// TIA Portal V18 export
// export: Created 2025-12-01T17:50:36.3947Z, ExportSetting None, DisplayName Totally Integrated Automation Portal, DisplayVersion V18 Update 5, DisplayName TIA Portal Openness, DisplayVersion V18 Update 5, DisplayName TIA Portal Teamcenter Gateway, DisplayVersion V18, DisplayName TIA Portal Version Control Interface, DisplayVersion V18, DisplayName STEP 7 Professional, DisplayVersion V18 Update 5, DisplayName STEP 7 Safety, DisplayVersion V18, DisplayName WinCC Professional, DisplayVersion V18 Update 5
DATA_BLOCK "AutoProcessData_Buffer_Clear"   // DB1602
{ S7_Optimized_Access := 'FALSE' }
// stored: AutoNumber false
   VAR RETAIN
      DataBuffer : Array[0..60] of "ProcessData";
      DataBufferClear : "ProcessData";
      VAL { S7_SetPoint := 'True'} : Int;
   END_VAR
BEGIN
END_DATA_BLOCK
